FUNCTION_BLOCK FB_AllMoversToStartpos
VAR_INPUT
	bXTS_MoveToStartPos		: BOOL;
	rInitPosition			: LREAL;
	rInitVelocity			: LREAL;
	rRailLength				: LREAL;
	rGap					: LREAL;
END_VAR

VAR_IN_OUT
	Mover					: ARRAY [*] OF AXIS_REF;
END_VAR

VAR
	i						: DINT;
	fbMoveToStartPos		: ARRAY [1..iMaxNumbMovers] OF MC_MoveRelativeCA;
END_VAR

// **************************************************************************************
// Move all Movers to initial position
// **************************************************************************************

FOR i:=1 TO UPPER_BOUND(Mover,1) DO
	
	IF Mover[i].NcToPlc.ModuloSetPos < (rInitPosition - 1) THEN
		fbMoveToStartPos[i].Distance := rInitPosition - Mover[i].NcToPlc.ModuloSetPos;
	ELSE;
		fbMoveToStartPos[i].Distance := rInitPosition - Mover[i].NcToPlc.ModuloSetPos + rRailLength ;
	END_IF
		
	fbMoveToStartPos[i](
		Axis			:= Mover[i], 
		Execute			:= bXTS_MoveToStartPos, 
		ContinuousUpdate:= TRUE, 
		Velocity		:= rInitVelocity, 
		Gap				:= rGap, 
		);

END_FOR

END_FUNCTION_BLOCK

(* stored: Version 1.1.0.1, ProductVersion 3.1.4024.12
   POU FB_AllMoversToStartpos: Id {6142d546-14f9-4e5d-adf3-1fbc5d04708e}, SpecialFunc None *)
